// Brief: Slave Arm Error Hold
FUNCTION_BLOCK PUBLIC FB_SlaveCtrlError EXTENDS FB_SlaveArmCtrlBase
VAR
	// velocity for full damping
	m_maxAdjustVel :Vec3d := [1.2, 1.2, 0.3];
	
	// velocity start to enable damping
	m_velLBForDamp :Vec3d := [1.0, 1.0, 0.2];
	
	// max damp
	m_maxDamp :Vec3d := [50, 50, 500];
	
	// distance buffer from joint limit to start damp
	m_limitBufferForDamp :Vec3d :=[20*g_deg2Rad, 20*g_deg2Rad, 0.03];
END_VAR

// override this function in each exact controller
METHOD PROTECTED calcCmdJntPos : BOOL
VAR_IN_OUT CONSTANT
	// endoscope pose in cart coordinate
	i_endoscopePose : ST_Frame;
	
	// master arm data
	i_masterStatus :ST_MasterStatus;
	
	// setup arm data
	i_setupStatus: ST_SetupStatus;
	
	// slave arm data
	i_slaveArm :FB_SlaveArm;
END_VAR
VAR
	i:INT;
END_VAR
m_cmdJntPos := i_slaveArm.curJntPos;
END_METHOD

// override this function in each exact controller
METHOD PROTECTED calcCmdJntTrq : BOOL
VAR_IN_OUT CONSTANT
	i_endoscopePose : ST_Frame;
	i_masterStatus :ST_MasterStatus;
	i_setupStatus: ST_SetupStatus;
	i_slaveArm :FB_SlaveArm;
END_VAR
VAR
	i :INT;
	dampScale :LREAL;
	limitDis :LREAL;
END_VAR
// set joint torque to zero in default
m_cmdJntTrq := g_zeroVec8d;

// enable joint adjust if its error is recoverable
FOR i:=1 TO 3 DO
	// disable joint
	IF NOT(i_slaveArm.adjustOn) THEN
		m_jntEnableFlag[i]:= 0;
		m_jntOPMode[i]:=DriverOPMode_Pos;
		CONTINUE;
	END_IF
	
	// enable joint
	m_jntEnableFlag[i]:= 1;
	m_jntOPMode[i]:=DriverOPMode_Trq;
	
	// add damp near joint limit
	IF (i_slaveArm.curJntPos[i] > GVL_SlaveMotorParameters.g_maxDHJntPos[i] - m_limitBufferForDamp[i] AND  i_slaveArm.curJntVel[i]> 0 ) 
		OR (i_slaveArm.curJntPos[i] < GVL_SlaveMotorParameters.g_minDHJntPos[i] + m_limitBufferForDamp[i] AND  i_slaveArm.curJntVel[i]<0 )  THEN
		limitDis := MIN(GVL_SlaveMotorParameters.g_maxDHJntPos[i] - i_slaveArm.curJntPos[i], i_slaveArm.curJntPos[i]-GVL_SlaveMotorParameters.g_minDHJntPos[i]);
		dampScale  :=LIMIT(0, 1-limitDis/m_limitBufferForDamp[i],1);
		m_cmdJntTrq[i]:= -dampScale * m_maxDamp[i] * i_slaveArm.curJntVel[i];
	END_IF

	// compute damp
	IF ABS(i_slaveArm.curJntVel[i]) > m_velLBForDamp[i] THEN 
		dampScale:=LIMIT(0, (ABS(i_slaveArm.curJntVel[i])- m_velLBForDamp[i])/(m_maxAdjustVel[i] - m_velLBForDamp[i]), 1 );
		m_cmdJntTrq[i] :=m_cmdJntTrq[i] -i_slaveArm.curJntVel[i] * m_maxDamp[i] * dampScale;
	END_IF

END_FOR
END_METHOD

// override this function in each exact controller
// NOTICE: set joint control mode here, and do some initialization if needed
METHOD PUBLIC init : BOOL
VAR_IN_OUT CONSTANT
	i_slaveArm	:FB_SlaveArm;
END_VAR
VAR_IN_OUT 
	r_slaveArmCtrlCmd :ST_SlaveArmCtrlCmds;
END_VAR


VAR
	i:INT;
END_VAR
SUPER^.Init(i_slaveArm,r_slaveArmCtrlCmd);

// disable first three joints
m_jntEnableFlag[1]:= 0;
m_jntEnableFlag[2]:= 0;
m_jntEnableFlag[3]:= 0;

// disable instrument joints which is in error 
//FOR i:=4 TO g_sJntNum DO
//	IF SafetyCheck.m_SafetyCheck.m_jntErrFlag[i_slaveArm.armIdx, i+g_setupJntNum, 2] OR  SafetyCheck.m_SafetyCheck.m_jntErrFlag[i_slaveArm.armIdx, i+g_setupJntNum, 3] THEN
//		m_jntEnableFlag[i] := 0;
//	ELSE
//		m_jntEnableFlag[i] := 1;
//	END_IF
//END_FOR
 
 // update commands to arm
copyCmds(r_slaveArmCtrlCmd);
END_METHOD

END_FUNCTION_BLOCK

(* stored: Version 1.1.0.1, ProductVersion 3.1.4024.12
   POU FB_SlaveCtrlError: Id {78b2e60d-537e-446e-8b3b-6db63d5ab02c}, SpecialFunc None
   Method calcCmdJntPos: Id {c2b94d3d-dd32-4b7a-a379-1afc098a58f1}
   Method calcCmdJntTrq: Id {fdc795ea-c7ad-49b5-ae7f-ec8937b0edfa}
   Method init: Id {e6a6f329-eae4-4e64-b8ba-0dd027b37a8e} *)
